FUNCTION_BLOCK E_MERGE_3 (* Composite Function Block Type *)
  (* Standard: 61499-2 *)
  (* Version 0.0, 9/22/2026, macie, Schneider Electric, template *)
  PACKAGE Main;
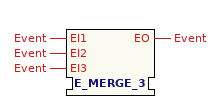
  EVENT_INPUT
    EI1; (* Initialization Request *)
    EI2; (* Normal Execution Request *)
    EI3;
  END_EVENT
  EVENT_OUTPUT
    EO; (* Initialization Confirm *)
  END_EVENT
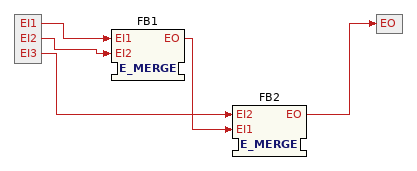
  FBS
    FB1 : E_MERGE;
    FB2 : E_MERGE;
  END_FBS
  EVENT_CONNECTIONS
    EI3 TO FB2.EI2;
    EI1 TO FB1.EI1;
    EI2 TO FB1.EI2;
    FB1.EO TO FB2.EI1;
    FB2.EO TO EO;
  END_CONNECTIONS
END_FUNCTION_BLOCK
